// TIA Portal project "Projeto Automação Industrial" (V15.1)
// Vorlageprojekt für das Buch mit Zielsystem S7-1200

(* hardware
DEVICE "S7-1200-Station_1"  S7-1200 Station
   slot 0: "Baugruppenträger_0"  Rack  V1.0
   slot 1: "PLC_1"  CPU 1211C DC/DC/DC  6ES7 211-1AE40-0XB0  V4.1
*)

// ===== PLC "PLC_1"  CPU 1211C DC/DC/DC =====

VAR_GLOBAL   // PLC tag table "Standard-Variablentabelle"
   "Esteira 1" AT %A0.0 : Bool;
   "Sensor de Saída" AT %E0.0 : Bool;
   "Botão Liga" AT %E0.1 : Bool;
   "Luz do Botão Liga" AT %Q1.1 : Bool;
   "Iniciar Processo" AT %Q3.0 : Bool;
   "Classificador 1" AT %Q2.1 : Bool;
   "Classificador 2" AT %Q2.2 : Bool;
   "Classificador 3" AT %Q2.3 : Bool;
   "Lâmina de Parada" AT %Q0.1 : Bool;
   "Classificador 1 Motor" AT %Q0.3 : Bool;
   "Classificador 1 Esteira" AT %Q0.4 : Bool;
   "Parar esteiras" AT %Q2.4 : Bool;
   "Sensor" AT %ID30 : DInt;
   "Contador 1" AT %QD30 : DInt;
   "Botão Desliga" AT %I0.3 : Bool;
   "Contador 1 Display" AT %Q2.5 : Bool;
   "Timer de Esteira" AT %Q2.6 : Bool;
   "Contador 2" AT %QD34 : DInt;
   "Contador 2 Display" AT %Q2.7 : Bool;
   "Contador 3" AT %QD38 : DInt;
   "Contador 3 Display" AT %Q1.4 : Bool;
   "Esteira 2" AT %Q0.2 : Bool;
   "Classificador 2 Motor" AT %Q0.5 : Bool;
   "Classificador 2 Esteira" AT %Q0.6 : Bool;
   "Classificador 3 Motor" AT %Q0.7 : Bool;
   "Classificador 3 Esteira" AT %Q1.0 : Bool;
   "Luz do Botão Desliga" AT %Q1.3 : Bool;
   "Retirada de Peça" AT %Q3.1 : Bool;
   "Tempo de Saída" AT %Q3.2 : Bool;
   "Reset" AT %I0.2 : Bool;
   "Luz do Botão de Reset" AT %Q1.2 : Bool;
END_VAR

// folder: System blocks/Program resources

DATA_BLOCK "IEC_Counter_0_DB"   // DB1
{ S7_Optimized_Access := 'TRUE' }
AUTHOR : Simatic
FAMILY : IEC
NAME : CNTR
VERSION : 1.0
// stored: InstanceOfName IEC_COUNTER
"IEC_COUNTER"
BEGIN
END_DATA_BLOCK

DATA_BLOCK "IEC_Timer_0_DB"   // DB2
{ S7_Optimized_Access := 'TRUE' }
AUTHOR : Simatic
FAMILY : IEC
NAME : IEC_TMR
VERSION : 1.0
// stored: InstanceOfName IEC_TIMER
"IEC_TIMER"
BEGIN
END_DATA_BLOCK

DATA_BLOCK "IEC_Timer_0_DB_4"   // DB3
{ S7_Optimized_Access := 'TRUE' }
AUTHOR : Simatic
FAMILY : IEC
NAME : IEC_TMR
VERSION : 1.0
// stored: InstanceOfName IEC_TIMER
"IEC_TIMER"
BEGIN
END_DATA_BLOCK

DATA_BLOCK "IEC_Counter_0_DB_1"   // DB5
{ S7_Optimized_Access := 'TRUE' }
AUTHOR : Simatic
FAMILY : IEC
NAME : CNTR
VERSION : 1.0
// stored: InstanceOfName IEC_COUNTER
"IEC_COUNTER"
BEGIN
END_DATA_BLOCK

DATA_BLOCK "IEC_Counter_0_DB_2"   // DB6
{ S7_Optimized_Access := 'TRUE' }
AUTHOR : Simatic
FAMILY : IEC
NAME : CNTR
VERSION : 1.0
// stored: InstanceOfName IEC_COUNTER
"IEC_COUNTER"
BEGIN
END_DATA_BLOCK

DATA_BLOCK "IEC_Timer_0_DB_2"   // DB7
{ S7_Optimized_Access := 'TRUE' }
AUTHOR : Simatic
FAMILY : IEC
NAME : IEC_TMR
VERSION : 1.0
// stored: InstanceOfName IEC_TIMER
"IEC_TIMER"
BEGIN
END_DATA_BLOCK

DATA_BLOCK "IEC_Timer_0_DB_1"   // DB8
{ S7_Optimized_Access := 'TRUE' }
AUTHOR : Simatic
FAMILY : IEC
NAME : IEC_TMR
VERSION : 1.0
// stored: InstanceOfName IEC_TIMER
"IEC_TIMER"
BEGIN
END_DATA_BLOCK

DATA_BLOCK "IEC_Timer_0_DB_3"   // DB9
{ S7_Optimized_Access := 'TRUE' }
AUTHOR : Simatic
FAMILY : IEC
NAME : IEC_TMR
VERSION : 1.0
// stored: InstanceOfName IEC_TIMER
"IEC_TIMER"
BEGIN
END_DATA_BLOCK

// folder: (top level)

FUNCTION "MHJ-PLC-Lab-Function-S71200" : Void   // FC9000, SCL
{ S7_Optimized_Access := 'TRUE' }
VERSION : 0.1
   VAR_TEMP
      rdTimeReturn : Int;
      outputTime : DTL;
      SyncVal : Byte;
      forVal : Int;
      forVal_2 : Int;
      Value : Byte;
   END_VAR
   VAR CONSTANT
      CompVal : Byte := 16#34;
      Value_01 : Byte := 16#11;
      Value_01_DW : DWord := 16#A165_D992;
      Value_02_DW : DWord := 16#58BE_4401;
   END_VAR
BEGIN

   #Value:=PEEK(area := 16#82,
        dbNumber := 0,
        byteOffset := 511);
   #Value := #Value + 1;

   POKE(area := 16#82,
        dbNumber := 0,
        byteOffset := 511,
        value := #Value);

   POKE(area:=16#81,
        dbNumber:=0,
        byteOffset:=1016,
        value:=#Value_01_DW);
   POKE(area := 16#81,
        dbNumber := 0,
        byteOffset := 1020,
        value := #Value_02_DW);

   POKE(area := 16#81,
        dbNumber := 0,
        byteOffset := 511,
        value := B#16#00);

   FOR #forVal := 0 TO 120 DO
       FOR #forVal_2:=0 TO 10 DO
           #rdTimeReturn:=RD_SYS_T(#outputTime);
           #rdTimeReturn := WR_SYS_T(#outputTime);
           #rdTimeReturn := RD_SYS_T(#outputTime);
           #rdTimeReturn := WR_SYS_T(#outputTime);
       END_FOR;
       #SyncVal:= PEEK(area := 16#81,
                      dbNumber := 0,
                      byteOffset := 511);
       IF #SyncVal = #CompVal THEN
          GOTO M_1;
       END_IF;
   END_FOR;
   RETURN;

   M_1:
   POKE(area := 16#81,
        dbNumber := 0,
        byteOffset := 511,
        value := B#16#0);
END_FUNCTION

ORGANIZATION_BLOCK "Main"   // OB1, LAD, ProgramCycle
TITLE = "Main Program Sweep (Cycle)"
{ S7_Optimized_Access := 'TRUE' }
VERSION : 0.1
   VAR_INPUT
      Initial_Call : Bool;   // Initial call of this OB
      Remanence : Bool;   // =True, if remanent data are available
   END_VAR
BEGIN

REGION Network 1: Konnektierungsbaustein für PLC-Lab
   // Im Netzwerk 1 wird der Konnektierungsbaustein für PLC-Lab aufgerufen.
   // Dieser Aufruf darf nicht entfernt werden!
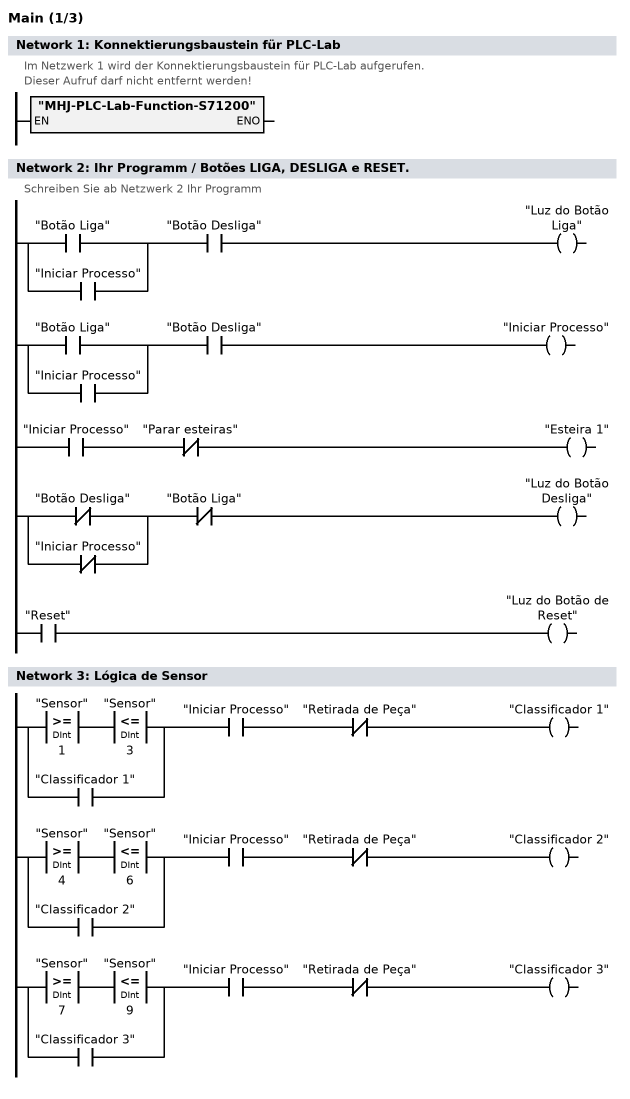
   RUNG wire#powerrail
      "MHJ-PLC-Lab-Function-S71200"()
   END_RUNG
   // the same network as SCL:
   "MHJ-PLC-Lab-Function-S71200"();
END_REGION

REGION Network 2: Ihr Programm / Botões LIGA, DESLIGA e RESET.
   // Schreiben Sie ab Netzwerk 2 Ihr Programm
   RUNG wire#powerrail
      Contact( "Botão Liga" )
      wire#w1
      Contact( "Botão Desliga" )
      Coil( "Luz do Botão Liga" )
   END_RUNG
   RUNG wire#powerrail
      Contact( "Iniciar Processo" )
   END_RUNG wire#w1
   RUNG wire#powerrail
      Contact( "Botão Liga" )
      wire#w2
      Contact( "Botão Desliga" )
      Coil( "Iniciar Processo" )
   END_RUNG
   RUNG wire#powerrail
      Contact( "Iniciar Processo" )
   END_RUNG wire#w2
   RUNG wire#powerrail
      Contact( "Iniciar Processo" )
      I_Contact( "Parar esteiras" )
      Coil( "Esteira 1" )
   END_RUNG
   RUNG wire#powerrail
      I_Contact( "Botão Desliga" )
      wire#w3
      I_Contact( "Botão Liga" )
      Coil( "Luz do Botão Desliga" )
   END_RUNG
   RUNG wire#powerrail
      I_Contact( "Iniciar Processo" )
   END_RUNG wire#w3
   RUNG wire#powerrail
      Contact( "Reset" )
      Coil( "Luz do Botão de Reset" )
   END_RUNG
   // the same network as SCL:
   "Luz do Botão Liga" := ("Botão Liga" OR "Iniciar Processo") AND "Botão Desliga";
   "Iniciar Processo" := ("Botão Liga" OR "Iniciar Processo") AND "Botão Desliga";
   "Esteira 1" := "Iniciar Processo" AND NOT "Parar esteiras";
   "Luz do Botão Desliga" := (NOT "Botão Desliga" OR NOT "Iniciar Processo") AND NOT "Botão Liga";
   "Luz do Botão de Reset" := "Reset";
END_REGION

REGION Network 3: Lógica de Sensor
   RUNG wire#powerrail
      { S7_Templates := "SrcType := DInt" } GE_Contact(in1 := "Sensor", in2 := 1)
      { S7_Templates := "SrcType := DInt" } LE_Contact(in1 := "Sensor", in2 := 3)
      wire#w1
      Contact( "Iniciar Processo" )
      I_Contact( "Retirada de Peça" )
      Coil( "Classificador 1" )
   END_RUNG
   RUNG wire#powerrail
      Contact( "Classificador 1" )
   END_RUNG wire#w1
   RUNG wire#powerrail
      { S7_Templates := "SrcType := DInt" } GE_Contact(in1 := "Sensor", in2 := 4)
      { S7_Templates := "SrcType := DInt" } LE_Contact(in1 := "Sensor", in2 := 6)
      wire#w2
      Contact( "Iniciar Processo" )
      I_Contact( "Retirada de Peça" )
      Coil( "Classificador 2" )
   END_RUNG
   RUNG wire#powerrail
      Contact( "Classificador 2" )
   END_RUNG wire#w2
   RUNG wire#powerrail
      { S7_Templates := "SrcType := DInt" } GE_Contact(in1 := "Sensor", in2 := 7)
      { S7_Templates := "SrcType := DInt" } LE_Contact(in1 := "Sensor", in2 := 9)
      wire#w3
      Contact( "Iniciar Processo" )
      I_Contact( "Retirada de Peça" )
      Coil( "Classificador 3" )
   END_RUNG
   RUNG wire#powerrail
      Contact( "Classificador 3" )
   END_RUNG wire#w3
   // the same network as SCL:
   "Classificador 1" := ((("Sensor" >= 1) AND ("Sensor" <= 3)) OR "Classificador 1") AND "Iniciar Processo" AND NOT "Retirada de Peça";
   "Classificador 2" := ((("Sensor" >= 4) AND ("Sensor" <= 6)) OR "Classificador 2") AND "Iniciar Processo" AND NOT "Retirada de Peça";
   "Classificador 3" := ((("Sensor" >= 7) AND ("Sensor" <= 9)) OR "Classificador 3") AND "Iniciar Processo" AND NOT "Retirada de Peça";
END_REGION

REGION Network 4: Ativação de Classificadores
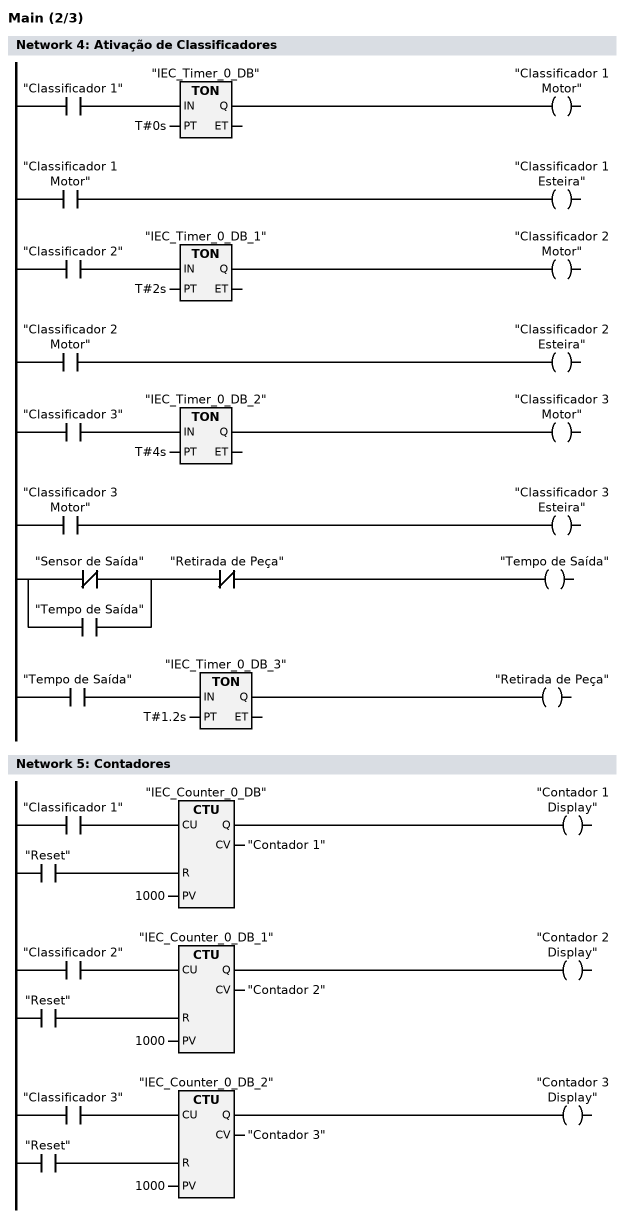
   "IEC_Timer_0_DB".TON(IN := "Classificador 1", PT := T#0s);
   "Classificador 1 Motor" := "IEC_Timer_0_DB".Q;
   "Classificador 1 Esteira" := "Classificador 1 Motor";
   "IEC_Timer_0_DB_1".TON(IN := "Classificador 2", PT := T#2s);
   "Classificador 2 Motor" := "IEC_Timer_0_DB_1".Q;
   "Classificador 2 Esteira" := "Classificador 2 Motor";
   "IEC_Timer_0_DB_2".TON(IN := "Classificador 3", PT := T#4s);
   "Classificador 3 Motor" := "IEC_Timer_0_DB_2".Q;
   "Classificador 3 Esteira" := "Classificador 3 Motor";
   "Tempo de Saída" := (NOT "Sensor de Saída" OR "Tempo de Saída") AND NOT "Retirada de Peça";
   "IEC_Timer_0_DB_3".TON(IN := "Tempo de Saída", PT := T#1.2s);
   "Retirada de Peça" := "IEC_Timer_0_DB_3".Q;
END_REGION

REGION Network 5: Contadores
   "IEC_Counter_0_DB".CTU(CU := "Classificador 1", R := "Reset", PV := 1000, CV => "Contador 1");
   "Contador 1 Display" := "IEC_Counter_0_DB".Q;
   "IEC_Counter_0_DB_1".CTU(CU := "Classificador 2", R := "Reset", PV := 1000, CV => "Contador 2");
   "Contador 2 Display" := "IEC_Counter_0_DB_1".Q;
   "IEC_Counter_0_DB_2".CTU(CU := "Classificador 3", R := "Reset", PV := 1000, CV => "Contador 3");
   "Contador 3 Display" := "IEC_Counter_0_DB_2".Q;
END_REGION

REGION Network 6: Parar a primeira esteira
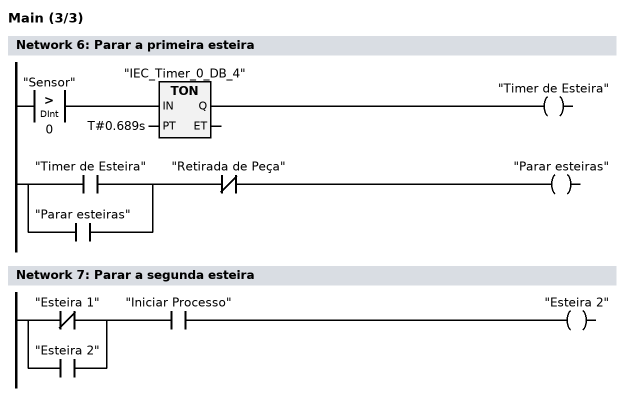
   "IEC_Timer_0_DB_4".TON(IN := "Sensor" > 0, PT := T#0.689s);
   "Timer de Esteira" := "IEC_Timer_0_DB_4".Q;
   "Parar esteiras" := ("Timer de Esteira" OR "Parar esteiras") AND NOT "Retirada de Peça";
END_REGION

REGION Network 7: Parar a segunda esteira
   RUNG wire#powerrail
      I_Contact( "Esteira 1" )
      wire#w1
      Contact( "Iniciar Processo" )
      Coil( "Esteira 2" )
   END_RUNG
   RUNG wire#powerrail
      Contact( "Esteira 2" )
   END_RUNG wire#w1
   // the same network as SCL:
   "Esteira 2" := (NOT "Esteira 1" OR "Esteira 2") AND "Iniciar Processo";
END_REGION
END_ORGANIZATION_BLOCK